FUNCTION_BLOCK FB_Homing
VAR_IN_OUT
	stAxis  	: ARRAY [GVL.cXP .. GVL.cXM] OF ST_AxisGroup;
	bTopEntry	: BOOL;
END_VAR
VAR_OUTPUT
	bBusy : BOOL;
END_VAR
VAR
	//state-machine
	nCurrentState	: INT;
	nNextState		: INT;

	//other var
	fbHomeDelay		: TON;
	
	//testVar
	a,b,c :INT;
END_VAR

//////////////////////////////////////////////////
//Performs homing routine						//
//////////////////////////////////////////////////

IF bTopEntry = TRUE THEN
	bTopEntry := FALSE;
	nNextState := 410;
	bBusy := TRUE;
END_IF	
nCurrentState := nNextState;
CASE nCurrentState OF
	0:
	
	410: //Clear Homed flag and calibrated flag
		fbHomeDelay(IN:=FALSE);
		stAxis[GVL.cXP].mcHome(Axis := stAxis[GVL.cXP].axisRef, HomingMode := MC_ResetCalibration, bCalibrationCam := TRUE, Execute := TRUE);
		stAxis[GVL.cXM].mcHome(Axis := stAxis[GVL.cXM].axisRef, HomingMode := MC_ResetCalibration, bCalibrationCam := TRUE, Execute := TRUE);
		stAxis[GVL.cXP].bIsCalibrated := FALSE;
		stAxis[GVL.cXM].bIsCalibrated := FALSE;
		IF stAxis[GVL.cXP].mcHome.Done AND stAxis[GVL.cXM].mcHome.Done THEN
			stAxis[GVL.cXP].mcHome(Axis := stAxis[GVL.cXP].axisRef, Execute := FALSE);
			stAxis[GVL.cXM].mcHome(Axis := stAxis[GVL.cXM].axisRef, Execute := FALSE);
			nNextState := 420;
			a:=a+1;
		END_IF
		b:=b+1;
		
	420: //Scan for home switch
		stAxis[GVL.cXP].mcJog(Axis := stAxis[GVL.cXP].axisRef, Mode := MC_JOGMODE_CONTINOUS, Velocity := GVL.cScanVel, JogBackwards := NOT stAxis[GVL.cXP].bLimitHome);
		stAxis[GVL.cXM].mcJog(Axis := stAxis[GVL.cXM].axisRef, Mode := MC_JOGMODE_CONTINOUS, Velocity := GVL.cScanVel, JogForward := NOT stAxis[GVL.cXM].bLimitHome);
		IF stAxis[GVL.cXP].bLimitHome AND stAxis[GVL.cXM].bLimitHome THEN
			stAxis[GVL.cXP].mcJog(Axis := stAxis[GVL.cXP].axisRef, Mode := MC_JOGMODE_CONTINOUS, JogBackwards := FALSE);
			stAxis[GVL.cXM].mcJog(Axis := stAxis[GVL.cXM].axisRef, Mode := MC_JOGMODE_CONTINOUS, JogForward := FALSE);
			nNextState := 430;
		END_IF

	430: //back off from switch
		stAxis[GVL.cXP].mcJog(Axis := stAxis[GVL.cXP].axisRef, Mode := MC_JOGMODE_CONTINOUS, Velocity := GVL.cScanVel, JogForward := stAxis[GVL.cXP].bLimitHome);
		stAxis[GVL.cXM].mcJog(Axis := stAxis[GVL.cXM].axisRef, Mode := MC_JOGMODE_CONTINOUS, Velocity := GVL.cScanVel, JogBackwards := stAxis[GVL.cXM].bLimitHome);
		IF NOT stAxis[GVL.cXP].bLimitHome AND NOT stAxis[GVL.cXM].bLimitHome THEN
			stAxis[GVL.cXP].mcJog(Axis := stAxis[GVL.cXP].axisRef, Mode := MC_JOGMODE_CONTINOUS, JogForward := FALSE);
			stAxis[GVL.cXM].mcJog(Axis := stAxis[GVL.cXM].axisRef, Mode := MC_JOGMODE_CONTINOUS, JogBackwards := FALSE);
			nNextState := 440;
		END_IF
		
	440: //slowly homed back to switch
		stAxis[GVL.cXP].mcJog(Axis := stAxis[GVL.cXP].axisRef, Mode := MC_JOGMODE_CONTINOUS, Velocity := GVL.cHomeVel, JogBackwards := NOT stAxis[GVL.cXP].bLimitHome);
		stAxis[GVL.cXM].mcJog(Axis := stAxis[GVL.cXM].axisRef, Mode := MC_JOGMODE_CONTINOUS, Velocity := GVL.cHomeVel, JogForward := NOT stAxis[GVL.cXM].bLimitHome);
		IF stAxis[GVL.cXP].bLimitHome AND stAxis[GVL.cXM].bLimitHome THEN
			stAxis[GVL.cXP].mcJog(Axis := stAxis[GVL.cXP].axisRef, Mode := MC_JOGMODE_CONTINOUS, JogBackwards := FALSE);
			stAxis[GVL.cXM].mcJog(Axis := stAxis[GVL.cXM].axisRef, Mode := MC_JOGMODE_CONTINOUS, JogForward := FALSE);
			nNextState := 450;
		END_IF	

	450://delay
		fbHomeDelay(IN:=TRUE, PT:=T#100MS);
		IF fbHomeDelay.Q THEN
			fbHomeDelay(IN:=FALSE);	
			nNextState := 460;
		END_IF
		
	460://set home
		stAxis[GVL.cXP].mcHome(Axis := stAxis[GVL.cXP].axisRef, Position := GVL.cPosStart, HomingMode := MC_DIRECT, Execute := TRUE);
		stAxis[GVL.cXM].mcHome(Axis := stAxis[GVL.cXM].axisRef, Position := GVL.cPosEnd, HomingMode := MC_DIRECT, Execute := TRUE);	
		IF stAxis[GVL.cXP].mcHome.Done AND stAxis[GVL.cXM].mcHome.Done THEN
			stAxis[GVL.cXP].mcHome(Axis := stAxis[GVL.cXP].axisRef, Execute := FALSE);
			stAxis[GVL.cXM].mcHome(Axis := stAxis[GVL.cXM].axisRef, Execute := FALSE);
			nNextState := 470;
		END_IF	
		
	470://delay
		fbHomeDelay(IN:=TRUE, PT:=T#100MS);
		IF fbHomeDelay.Q THEN
			fbHomeDelay(IN:=FALSE);	
			nNextState := 480;
		END_IF
		
	480: //End Action
		bBusy := FALSE;
		nNextState :=0;
END_CASE

END_FUNCTION_BLOCK

(* stored: Version 1.1.0.1, ProductVersion 3.1.4020.12
   POU FB_Homing: Id {67eb6d7f-00ee-47b8-9057-855207043b52}, SpecialFunc None *)
